{attribute 'qualified_only'}
VAR_GLOBAL
	bMotorsInitialized : BOOL;
	sMotorInitState : STRING;
	bPageChange : BOOL;
	bLftColumnsLatched : BOOL;
	bRhtColumnsLatched : BOOL;
	
	///////////////////// SAFETY /////////////////////////////////
	bRunSafety			AT %Q* : BOOL := TRUE; 	// Used to run safety program
	bSafetyErrorAck 	AT %Q* : BOOL; 			// Sequence to acknowledge safety error : False > True > False.
	bSafetyBypass		AT %Q* : BOOL;			//Used to Bypass entire safety PLC. Should Only be accessible with high level credentials. 
	bSafetyOk 			AT %I* : BOOL;			// Safety protocol enacted 
	bFbRun 				AT %I* : BOOL;			// Safety Function Blocks are running
	bInRun				AT %I* : BOOL;			// Safety Program is Running
	bFbErr				AT %I* : BOOL;			// A Safety Function Block contains an error
	bComErr				AT %I* : BOOL;			// Safety program communication error
	bOtherErr			AT %I* : BOOL;			// Other safety error exist. (EDM FB)
	bTestErr			AT %I* : BOOL;
	
	bSafetyInit : BOOL;
	nPageIndex: INT;
	nPrevPageIndex: INT;
	bMotorInitFailedDisp: BOOL;
	bMuteSafety: BOOL;
	
	////////////////////////ERROR HANDLING//////////////////////
	motorErrorList	: E_motorErrorList;
	bErrorPresent 	: BOOL;
	bDispErrorIcon 	: BOOL;
	
	///////////////////////SETTINGS SCREEN//////////////////////
	sEditMessage	: STRING(1024) := 'Changing this value will effect program parameters. Only change this value if you understand what effect this will have.';
	sEditTitle 		: STRING := 'CAUTION';
	sDescTitle		: STRING := 'Description';
	sConvHeightMsg 	: STRING(1024) := 'Table height from ground to top of table to recieve spa from conveyor';
	sClampHeightMsg : STRING(1024) := 'Table height from ground to top of table so that spa lip is even with clamp frame for centering'; 
	sDownHeightMsg : STRING(1024) := 'Table height from gount to top of table when the table is all the way down';
	sCenterTorqueMsg : STRING(1024) := 'Torque width motors move to when centering the spa';
	sClampOnTorqueMsg : STRING(1024) := 'Torque clamp motors use when clamping onto spa lip';
	sClampOpenDistMsg : STRING(1024) := 'Distance between clamp frame jaws when opened all the way';
	sLftRotHomeSetMsg : STRING(1024) := 'Offset counts set on the motor when homing is complete';
	sRhtRotHomeSetMsg : STRING(1024) := 'Offset counts set on the motor when homing is complete';
	
	// === ERROR LOGGING ===
	aErrorData				: ARRAY[1..5,1..23] OF STRING;
	nErrorDataRow			: INT := 1;
	//Custom Errors
	sBlock	: STRING;
	sLoc	: STRING;
	nID		: UDINT;
	sMsg 	: STRING;
	
	bFlashSaveBtn 	: BOOL;
	bSaveBtnFlashOn : BOOL;
	bSaveBtn 		: BOOL;
	
	bResetMachine: BOOL;
END_VAR

(* stored: Version 1.1.0.1, ProductVersion 3.1.4024.13
   GVL GVL_machine: Id {a0afb58b-55f6-45c1-aaa9-7c62110c2d93} *)
